# EPICS substitutions: TEKMSO58LPApp/Db/devmso58lp.substitutions
file dev_msoxx.template
{
    pattern {P,     PORT, }
    {$(P),$(PORT)}
}
